PROGRAM INTERNAL _ToDo

(*
DESCRIPTION:
- _				DONE
- Arg			DONE 
- Broadcast		DONE
- Callable		DONE
- Dbg			DONE
- Ec			DONE
- Iter			DONE
- Result		DONE
- Runtime		DONR
- State			
- Strings		DONE
- Tags			DONE
*)

END_PROGRAM

(* stored: Version 1.1.0.1
   POU _ToDo: Id {98d49df4-7f63-4c32-911d-1781c23c5b9e}, SpecialFunc None *)
